FUNCTION_BLOCK FB_DehumidifySFC

VAR_OUTPUT
	SFCCurrentStep	:	STRING;
END_VAR
VAR_IN_OUT
	//IPSState					:	ST_InternalPowerStatus;
	IPSDemand					:	ST_PowerDemand;
	ConditioningRequirements	: 	ST_ConditioningRequirements;
	Control						:	ST_CoolingSystem_Control;
	Get							:	ST_CoolingSystemGet;	
END_VAR
VAR_OUTPUT
	SFCActive	:	BOOL;
END_VAR

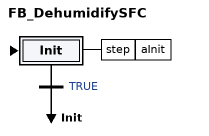
INITIAL_STEP Init:
    aInit(N);  // step action
END_STEP
TRANSITION FROM Init TO Init
    := TRUE;
END_TRANSITION

ACTION aInit:
SFCActive := False;
END_ACTION

METHOD SFCEnable : BOOL
VAR_INPUT
	Enable	:	Bool;
END_VAR
IF Enable THEN
	SFCInit := FALSE;
ELSE
	SFCActive:= FALSE;
	SFCInit := TRUE;
END_IF
END_METHOD

END_FUNCTION_BLOCK

(* stored: Version 1.1.0.1, ProductVersion 3.1.4024.12
   POU FB_DehumidifySFC: Id {97d87e63-d49b-4217-bef1-4cba729dec37}, SpecialFunc None
   Action aInit: Id {7339d1f3-fb31-43f1-99ca-ab7fa8a4cec1}
   Method SFCEnable: Id {a219cfa1-7553-4cb5-9a91-d25985d93a8c} *)
